Staubli VAL3: Day7.pjx

--- Day7.pjx ---
Parameters version=s8.13.1Cs9_BS2800 stackSize=5000 millimeterUnit=true
Program file=calc_fuel.pgx
Program file=start.pgx
Program file=stop.pgx
Data file=Day7.dtx
Library alias=util path=Disk://helpers/helpers.pjx
Library alias=math path=Disk://math/math.pjx
Library alias=str path=Disk://string/string.pjx
Library alias=stat path=Disk://statistics/statistics.pjx
Type name=lists path=Disk://types/lists/lists.pjx

--- Day7.dtx ---
string sInput
num nInput
lists lResult
  [0]
    string sString
num nResult
num nInput2
num nCounter[9]
num nResult2
num nInput1
num nMedian
num nDiff
num nRange
num nSum
num nDiffGuess
num nFuel

--- start.pgx ---
program start()
  local num l_nElement
  local num l_nString
  local num l_nCounter
  local num l_nResult
  local num l_nGuess
  local num l_nDiff
  local num l_nFuel
begin

  // read file
  call util:readFile("Disk://input_day7_test.txt", sInput)
  // sInput[0] = "1101,1,29,67,1102,....."

  call str:splitString(sInput,",", lResult)

  for l_nElement = 0 to size(lResult)-1

    // check for empty strings
    for l_nString = 0 to size(lResult[l_nElement].sString)-1
      if lResult[l_nElement].sString[l_nString] == ""
        delete(lResult[l_nElement].sString[l_nString])
      endIf
    endFor

    if l_nElement%2 == 0
      call util:vec2num(lResult[l_nElement].sString, nInput1)
    else
      call util:vec2num(lResult[l_nElement].sString, nInput2)
    endIf

    if l_nElement == 1
      call util:mergeVectors(nInput1,nInput2, nResult)
    elseIf l_nElement >=2
      if l_nElement % 2 == 0
        call util:mergeVectors(nResult,nInput1, nResult2)
      else
        call util:mergeVectors(nResult2,nInput2, nResult)
      endIf

    endIf
  endFor

  // PUZZLE 1
  // calculate median
  call stat:getMedian(nResult2, nMedian)

  // calculate difference to median and sum the differences up -> l_nResult
  resize(nDiff,1,size(nResult2))
  for l_nElement = 0 to size(nResult2)-1
    nDiff[l_nElement] = abs(nResult2[l_nElement] - nMedian)
  endFor

  call math:sum(nDiff, l_nResult)

  call util:printNum(l_nResult)
  // 344735

  // PUZZLE 2
//  resize(nFuel,1,10)
//  resize(nDiffGuess,1,11)
//  for l_nGuess = 0 to 999 step 10
//    if l_nGuess %10 == 0
//      ? l_nGuess
//    endIf

//    for l_nElement = 0 to size(nResult2)-1
//      l_nDiff = abs(nInput1[l_nElement] - l_nGuess)
//      call calc_fuel(l_nDiff,nFuel[l_nElement])
//    endFor

//    call math:sum(nFuel,nDiffGuess[l_nGuess/10])
//  endFor


end

--- calc_fuel.pgx ---
program calc_fuel(num x_nDiff, num& x_nFuel)
begin

  call util:range(0,x_nDiff+1,1,nRange)
  call math:sum(nRange, x_nFuel)

end
